PROGRAM P_Boiler
VAR
	bBoilerOn		: BOOL;
	bBoilerOff		: BOOL;
	bVBoilerSwitch	: BOOL;
	fbOnOffBoiler	: FB_OnOffLight;
END_VAR

fbOnOffBoiler(
	bSwitch:= bVBoilerSwitch OR bAdsBoilerOnOff,
	bOn:= bBoilerOn OR (todWinTime = tod#13:00 AND P_Temperatures.rTempBoiler < 55),
	bOff:= bBoilerOff,
	bAutoOff:= TRUE,
	tAutoOffTime:= t#4h,
	bLightNovRam:= bNovRamBoiler,
	bLightImpulsRelais=> bRelaisBoiler);

bAdsBoilerState := bNovRamBoiler;

END_PROGRAM

(* stored: Version 1.1.0.1
   POU P_Boiler: Id {d6afd0fa-1a48-43c8-91c7-a75759ddbc32}, SpecialFunc None *)
